Staubli VAL3: sendComplete.pgx

program sendComplete()
  local num buffer[2]
begin
  buffer[0] = MAGIC_HEADER
  buffer[1] = 2
  sioSet(socket, buffer)
end
